// TIA Portal V18 export
DATA_BLOCK "Emergency_Block_DB"   // DB2
VERSION : 0.1
// stored: AutoNumber true, InstanceOfName Emergency_Block, InstanceOfType FB
"Emergency_Block"
   // VAR_OUTPUT
   //    emergency_state : Bool;
   // END_VAR
BEGIN
END_DATA_BLOCK
